TYPE MastLight :
STRUCT
	Light1Color: cMastLightColor;  //Bottom Light
	Light1Appearance: cMastLightAppearance; //Bottom Light
	Light2Color: cMastLightColor;  //2nd From Bottom Light
	Light2Appearance: cMastLightAppearance;  //2nd From Bottom Light
	Light3Color: cMastLightColor;  //Center Light
	Light3Appearance: cMastLightAppearance; //Center Light
	Light4Color: cMastLightColor;  //2nd From Top Light
	Light4Appearance: cMastLightAppearance;  //2nd From Top Light
	Light5Color: cMastLightColor; //Top Light
	Light5Appearance: cMastLightAppearance; //Top Light
	MastBuzzerSW: BOOL; //On-Off Siwtch
	MastBuzzerSound: cMastLightBuzzerStyle; //Sound of the buzzer
	
END_STRUCT
END_TYPE

(* stored: Version 1.1.0.1, ProductVersion 3.1.4024.6
   DUT MastLight: Id {8d5f6505-aa4e-4783-9d70-b34fd5c6c9cb} *)
